PROGRAM Runner2
VAR
    foo : Foo;
    usesFoo : UsesFoo2;
END_VAR

usesFoo(foo:=foo);

END_PROGRAM

(* stored: Version 1.1.0.1, ProductVersion 3.1.4024.4
   POU Runner2: Id {7ad7e81d-b912-4142-80f3-89c4d7e1df8e}, SpecialFunc None *)
